FUNCTION_BLOCK ABSTRACT A_Actuator
VAR_INPUT
	
END_VAR
VAR_OUTPUT
END_VAR
VAR
	eCmd : E_ActuatorCmdType;
	
END_VAR

PROPERTY cmd : E_ActuatorCmdType
GET
cmd := eCmd;
END_GET
SET
eCmd := cmd;
executeCmd();
END_SET
END_PROPERTY

METHOD ABSTRACT executeCmd : BOOL
VAR_INPUT
	
END_VAR
END_METHOD

END_FUNCTION_BLOCK

(* stored: Version 1.1.0.1, ProductVersion 3.1.4024.2
   POU A_Actuator: Id {b488df22-3d2b-4774-a814-84ef0eeaf8f0}, SpecialFunc None
   Property cmd: Id {0a14cf9d-cb7b-4387-98fe-2a921e16e16c}
   Get Get: Id {27613634-6e42-4baa-a259-facd539ef149}
   Set Set: Id {dac50c59-5c61-457f-8380-6703eac5b669}
   Method executeCmd: Id {e220fc82-af7d-4a2a-a881-5e700ba87631} *)
